Universal Robots PolyScope program: TEST_SUB_106C.urp

Program TEST_SUB_106C (installation=GD directory=/programs/GD createdIn=5.13.0 lastSavedIn=5.13.0 robotSerialNumber=20205000017)
Calibrated DH parameters: a=[-0.000157, -0.56303, -0.236706, -0.000074, -0.000109, 0]; d=[0.181705, 47.632387, 369.599619, -417.058513, 0.119878, 0.115667]; alpha=[1.570881, -0.005074, -0.001247, 1.56886, -1.570997, 0]; deltaTheta=[0, -0.405485, 5.544791, 1.143886, -0.000009, -0.000001]
InitVariablesNode
BeforeStart
  prg_no := 0
  Script file /programs/GD/CONTROL/ALIGN_AXIS.script
    | def GET_NORM_VEC(p,axis=2):
    |   rot=p[0.0, 0.0, 0.0, p[3], p[4], p[5]]
    |   vec=p[0.0, 0.0, 0.0, 0.0, 0.0, 0.0]
    |   vec[axis]=1.0
    |   norm_p=pose_trans(rot,vec)
    |   return [norm_p[0], norm_p[1], norm_p[2]]
    | end
    | 
    | def GET_INNER_PRODUCT(v1,v2):
    |   return v1[0]*v2[0]+v1[1]*v2[1]+v1[2]*v2[2]
    | end
    | def GET_OUTER_PRODUCT(v1,v2):
    |   x=v1[1]*v2[2]-v1[2]*v2[1]
    |   y=v1[2]*v2[0]-v1[0]*v2[2]
    |   z=v1[0]*v2[1]-v1[1]*v2[0]
    |   return [x,y,z]
    | end
    | def GET_THETA(v1,v2):
    | #  cos=GET_INNER_PRODUCT(v1,v2) / norm(v1) / norm(v2)
    |   cos=GET_INNER_PRODUCT(v1,v2)
    |   g_cos=cos
    |   theta=norm(acos(cos))
    |   return theta
    | end
    | 
    | def GET_ALIGNED_POSE(target,feature,axis=2):
    |   feature_from_target=pose_trans(pose_inv(target),feature)
    |   g_f_from_t=feature_from_target
    |   nz_feature_from_target=GET_NORM_VEC(feature_from_target,axis)
    |   g_nz_f_from_t=nz_feature_from_target
    |   nz_target_from_target=[0.0, 0.0, 0.0]
    |   nz_target_from_target[axis]=1.0
    |   g_nz_t_from_t=nz_target_from_target
    | 
    |   theta=GET_THETA(nz_feature_from_target,nz_target_from_target)
    |   g_theta=theta
    |   rot_vec_n=normalize(GET_OUTER_PRODUCT(nz_target_from_target,nz_feature_from_target))
    | 
    |   if theta>d2r(90.0):
    |     theta=theta-d2r(180.0)
    |   end
    |   rot_vec=rot_vec_n * (theta)
    |   rot_p=p[0.0,0.0,0.0,rot_vec[0],rot_vec[1],rot_vec[2]]
    |   return pose_trans(target,rot_p)
    | end
    | def GET_ALIGNED_TCP(feature,axis=2):
    |   tcp=get_actual_tcp_pose()
    |   return GET_ALIGNED_POSE(tcp,feature,axis)
    | end
  Script file /programs/GD/CONTROL/CYCLE_CONTROL.script
    | def GET_REG(prg_no):
    |   WorkPosNo=read_input_integer_register(4)-1                       # GPII_WorkPosNo
    |   CaptIndex[WorkPosNo]=read_input_integer_register(21)-1           # GPII_CaptColNo
    |   CaptRowNo=read_input_integer_register(20)-1        # GPII_CaptRowNo
    |   CaptStepZ=read_input_integer_register(6) / 1000.0         # GPII_CaptStepZ
    |   ReCaptNo=0
    |   if (prg_no==1203):
    |     ReCaptNo=read_input_integer_register(22)                # GPII_ReCaptNo
    |   end
    |   ReCaptZ=read_input_integer_register(7) / 1000.0         # GPII_ReCaptZ
    |   CutOffZDef=read_input_integer_register(11) / 1000.0          # GPII_CutOffZ
    |   CrankDepthFull=read_input_integer_register(10) / 1000.0   # GPII_FullDepth
    | end
    | 
    | def POSE_SUB(p, teach_frame):
    |   return pose_trans(inv(teach_frame), p)
    | end
    | 
    | def GET_BUCKET_UPPER(pos=0):
    |   if UseNewCaptPos:
    |     p=POSE_SUB(CaptPoint_C, BucketM)
    |     pX=[BKWidth/2,CaptPointL_dX,BKWidth-CaptPointR_dX]
    |     p[0]=pX[pos]
    |   else:
    |     captpos=[CaptPoint_C,CaptPoint_L,CaptPoint_R]
    |     p=captpos[pos]
    |     p=POSE_SUB(p, BucketM)
    |   end
    |   return p
    | end
    | 
    | def SET_BUCKET_DEF():
    |   BucketM=pBucketM
    |   if (WorkPosNo<0):
    |     Bucket=pBucketC
    |   else:
    |     Bucket=pBucket[WorkPosNo]
    |   end
    | end
    | 
    | def SET_BUCKET():
    |   SET_BUCKET_DEF()
    |   Bucket[2]=Bucket[2]-CaptStepZ*CaptRowNo
    | end
    | 
    | def SET_CV():
    |   CV=pCV
    | end
    | 
    | def SET_CAPT_INDEX():
    |   CaptIndexWk=CaptIndex[WorkPosNo]
    |   ReCaptZWk=0
    |   if (prg_no==1203):
    |     if   (ReCaptNo==0):
    |       if (CaptIndexWk==0):
    |         if (0<=DistPillarBak):
    |           CaptIndexWk=1
    |         else:
    |           CaptIndexWk=2
    |         end
    |         ReCaptZWk=0
    |       else:
    |         CaptIndexWk=0
    |         ReCaptZWk=0
    |       end
    |     elif (ReCaptNo==1):
    |       if (CaptIndexWk==0):
    |         CaptIndexWk=0
    |         ReCaptZWk=-ReCaptZ
    |       else:
    |         CaptIndexWk=CaptIndexWk
    |         ReCaptZWk=-ReCaptZ
    |       end
    |     else:
    |       if (CaptIndexWk==0):
    |         CaptIndexWk=0
    |         ReCaptZWk=ReCaptZ
    |       else:
    |         CaptIndexWk=CaptIndexWk
    |         ReCaptZWk=ReCaptZ
    |       end
    |     end
    |   end
    | end
    | 
    | def GET_CAPTPOS():
    |   SET_BUCKET()
    |   SET_CAPT_INDEX()
    |   if UseNewCaptPos:
    |     p=GET_BUCKET_UPPER(CaptIndexWk)
    |     p[2]=p[2]-ReCaptZWk
    |   else:
    |     captpos=[CaptPoint_C,CaptPoint_L,CaptPoint_R]
    |     p=captpos[CaptIndexWk]
    |     p[2]=p[2]-ReCaptZWk
    |     p=POSE_SUB(p, BucketM)
    |   end
    |   return p
    | end
    | 
    | def CHECK_CAPTPOS():
    |   isOK=((CaptStepZ*(read_input_integer_register(20)-1)) < (read_input_integer_register(9) / 1000.0))
    |   return isOK
    | end
    | 
    | def GET_ZSLIDE_POS(p):
    |   p[2]=p[2]-CaptStepZ*CaptRowNo
    |   return p
    | end
    | 
    | def END_CYCLE():
    |   stopl(1.2)
    |   end_force_mode()
    |   end_freedrive_mode()
    |   socket_close(socket_name)
    | end
    | 
    | def CHECK_SPEED(smax,f=[1,1,1,1,1,1]):
    |   s=TCPSpeed
    |   i=0
    |   while (i<6):
    |     if ((f[i]==1) and (smax[i]<s[i])):
    |       return False
    |     end
    |     i=i+1
    |   end
    |   return True
    | end
  Script file /programs/GD/CONTROL/ZONE_CONTROL.script
    | def GET_DIST(P1, P2):
    |   return pose_dist(P1, P2)
    | end
    | def CHECK_DIST_NEAR(P1, P2, th):
    |   return (GET_DIST(P1, P2) < th)
    | end
    | def DIST_HOME():
    |   return pose_dist(gHome_Position,CurrPos_p)
    | end
    | 
    | def CHECK_HOME():
    |   return (DIST_HOME()<ZoneDistTh)
    | end
    | 
    | def DIST_CVUpper():
    |   if (read_input_integer_register(4)==1):
    |     p=g2GD_pos1
    |   else:
    |     p=g1GD_pos1
    |   end
    |   return pose_dist(p,CurrPos_p)
    | end
    | 
    | def CHECK_CVUpper():
    |   return (DIST_CVUpper()<ZoneDistTh)
    | end
    | 
    | def CHECK_RB_POS(prg_no):
    |   ret=True
    |   if (prg_no==1001):
    |     ret=CHECK_EVAC()
    |   end
    |   if ((prg_no==1201) or (prg_no==1401) or (prg_no==1402) or (prg_no==6001) or (prg_no==6101) or (prg_no==6401) or (prg_no==6102) or (prg_no==7001)):
    |     ret=CHECK_HOME()
    |   end
    |   if ((prg_no==1002) or (prg_no==1241) or (prg_no==1261)):
    |     ret=CHECK_BKInside()
    |   end
    |   if (prg_no==1251):
    |     ret=(CHECK_HOME() or CHECK_CVUpper())
    |   end
    |   if (ret != True):
    |     SubPrgResult=801
    |     sleep(999999.0)
    |   end
    | end
    | 
    | def DIST_ORIGIN():
    |   p=CurrPos_p
    |   o=p
    |   o[0]=0.0
    |   o[1]=0.0
    |   return pose_dist(o,p)
    | end
    | 
    | def CHECK_EVAC_ORG():
    |   return (EvacRadiusTh<DIST_ORIGIN())
    | end
    | 
    | def CHECK_EVAC_X():
    |   return (EvacXTh[0]<CurrPos_p[0] and CurrPos_p[0]<EvacXTh[1])
    | end
    | 
    | def CHECK_EVAC_Y():
    |   return (EvacYTh[0]<CurrPos_p[1] and CurrPos_p[1]<EvacYTh[1])
    | end
    | 
    | def CHECK_EVAC_Z():
    |   return (EvacZTh[0]<CurrPos_p[2])
    | end
    | 
    | def CHECK_EVAC():
    |   ret=True
    |   ret=(ret and CHECK_EVAC_ORG())
    |   ret=(ret and CHECK_EVAC_X())
    |   ret=(ret and CHECK_EVAC_Y())
    |   ret=(ret and CHECK_EVAC_Z())
    |   return ret
    | end
    | 
    | def CHECK_BKInside():
    |   ret=True
    |   pos=read_input_integer_register(4)
    |   if (pos>2):
    |     ret=False
    |   else:
    |     if (not read_input_boolean_register(13+pos)):
    |       ret=False
    |       ver_3=read_input_boolean_register(13+pos)
    |     else:
    |       bk=pBucket[pos-1]
    |       if (pos==1):
    |         ret=(ret and CurrPos_p[0]>ZoneHomeX)
    |         ret=(ret and bk[1]-(BucketWidth-ZoneBucketGap)<CurrPos_p[1] and CurrPos_p[1]<bk[1]-ZoneBucketGap)
    |       elif (pos==2):
    |         ret=(ret and CurrPos_p[0]<-ZoneHomeX)
    |         ret=(ret and bk[1]+ZoneBucketGap<CurrPos_p[1] and CurrPos_p[1]<bk[1]+(BucketWidth-ZoneBucketGap))
    |       end
    |     end
    |   end
    |   return ret
    | end
    | 
    | def CHECK_CVOutside():
    |   ret=True
    |   ret=(ret and gCV_11_M[0]-Zone6ThX<CurrPos_p[0])
    |   ret=(ret and CurrPos_p[0]<gCV_11_M[0]+Zone6ThX)
    |   ret=(ret and gCV_11_M[1]-Zone6ThY<CurrPos_p[1])
    |   ret=(ret and CurrPos_p[1]<gCV_11_M[1]+Zone6ThY)
    |   return (not ret)
    | end
    | 
    | def CHECK_ZONE(no):
    |   if (no==1):
    |     return (CurrPos_p[2]>=Zone1ZTh)
    |   elif (no==2):
    |     return (CurrPos_p[0]>ZoneHomeX)
    |   elif (no==3):
    |     return (CurrPos_p[0]<-ZoneHomeX)
    |   elif (no==4):
    |     return CHECK_CVUpper()
    |   elif (no==5):
    |     return CHECK_BKInside()
    |   elif (no==6):
    |     return CHECK_CVOutside()
    |   end
    | end
  Script file /programs/GD/CONTROL/ROTATE_CONTROL.script
    | def GET_TCP_FORCE_TOOL():
    |   force_torque=get_tcp_force()
    |   force_B=p[force_torque[0], force_torque[1], force_torque[2], 0, 0, 0]
    |   torque_B=p[force_torque[3], force_torque[4], force_torque[5], 0, 0, 0]
    |   tcp=get_actual_tcp_pose()
    |   rotation_BT=p[0, 0, 0, tcp[3], tcp[4], tcp[5]]
    |   force_T=pose_trans(pose_inv(rotation_BT), force_B)
    |   torque_T=pose_trans(pose_inv(rotation_BT), torque_B)
    |   force_torque_T=p[force_T[0], force_T[1], force_T[2], torque_T[0], torque_T[1], torque_T[2]]
    |   return force_torque_T
    | end
    | 
    | def CHECK_VALUE_RZ():
    |   return True
    | end
    | 
    | def GET_FORCE_VALUE_RZ(target):
    |   PoseSub= pose_sub (CurrPos_p,target)
    |   RYSub=r2d(PoseSub[4])
    |   RZSub=r2d(PoseSub[5])
    | #  if (RYSub<RZSupRYRange[0] or RZSupRYRange[1]<RYSub):
    | #    RZSupForceVal=0.0
    | #    return RZSupForceVal
    | #  end
    |   if (RZSub<0):
    |     RZMin=RZSupDegMin[0]
    |     RZRatio=RZSupRatio[0]
    |     RZOffset=RZSupOffset[0]
    |   else:
    |     RZMin=RZSupDegMin[1]
    |     RZRatio=RZSupRatio[1]
    |     RZOffset=-RZSupOffset[1]
    |   end
    |   if (norm(RZSub) >= norm(RZMin)):
    |     RZSupForceVal=(RZMin-RZSub)*RZRatio+RZOffset
    |   else:
    |     RZSupForceVal=0
    |   end
    |   if (RZSupForceVal<RZSupForceRange[0]):
    |     RZSupForceVal=RZSupForceRange[0]
    |   elif (RZSupForceRange[1]<RZSupForceVal):
    |     RZSupForceVal=RZSupForceRange[1]
    |   end
    |   if (RYSub<RZSupRYRange[0] or RZSupRYRange[1]<RYSub):
    |     RZSupForceVal=0
    |   end
    |   if ((not UseRZSupStep1) and (ForceStep==1)):
    |     RZSupForceVal=0
    |   end
    |   return RZSupForceVal
    | end
    | 
    | def GET_CVCORR_VALUE(target):
    |   PoseSub=pose_sub(CurrPos_p,target)
    |   RYSub=r2d(PoseSub[4])
    |   CVCorrRYSub=RYSub
    |   if (RYSub<0):
    |     RYMin=-CVCorrDegMin[0]
    |     RZRatio=CVCorrRatio[0]
    |     RZOffset=-CVCorrOffset[0]
    |   else:
    |     RYMin=-CVCorrDegMin[1]
    |     RZRatio=CVCorrRatio[1]
    |     RZOffset=CVCorrOffset[1]
    |   end
    |   if (norm(RYSub) >= norm(RYMin)):
    |     t=get_tcp_offset()
    |     CVCorrYVal=-t[2]*sin(d2r(RYSub))
    |     CVCorrRZVal=RYSub*RZRatio+RZOffset
    |   else:
    |     CVCorrYVal=0
    |     CVCorrRZVal=0
    |   end
    | end
    | 
    | def GET_CVCORR_POS(target):
    |   pos= pose_add (p[0,0,0,0,0,d2r(-CVCorrRZVal)],p[0,0,0,target[3],target[4],target[5]])
    |   pos=p[target[0],target[1],target[2],pos[3],pos[4],pos[5]]
    |   return pos
    | end
Robot Program (runOnlyOnce=true)
  SuppressedNode
    Wait Sleep waitTime=20
  If UseCutOffTCP
    Set NoAction tcp=TCP_1
    CutOffPos := p[0.,0.,0.,0.,0.,0.]
    CutOffPos := GET_ALIGNED_TCP(CutOffPos)
    Script: CurrPos=get_actual_tool_flange_pose()
    CutOffTCP := pose_trans(pose_inv(CurrPos),CutOffPos)
    SuppressedNode
      MoveJ speed 60 deg/s, acceleration 80 deg/s^2 (useActiveTCP=true) feature=Base
        Waypoint Variable (Variable): variable=CutOffPos
    Set NoAction tcp=ZERO
    CutOffTCP := pose_trans(get_tcp_offset(),CutOffTCP)
    Set NoAction tcp=TCP_1
  Else 
    Set NoAction tcp=TCP_1
    CutOffTCP := get_tcp_offset()
  Script: set_tcp(CutOffTCP)
  MoveL speed 250 mm/s, acceleration 50 mm/s^2 (useActiveTCP=true) feature=Base
    If UseZSlide
      gGD_pos5 := GET_ZSLIDE_POS(g1GD_pos5_NEAR)
    Else 
      gGD_pos5 := g1GD_pos5
    SuppressedNode
      Folder CV_CORR_RZ
        If UseCVCorr
          RZSub := CVCorrRZVal
          Set NoAction tcp=TCP_1
          Wait Sleep waitTime=0.02
          SuppressedNode
            Script: CurrPos_p=get_actual_tcp_pose()
          Script: CurrPos_p=gGD_pos5
          SuppressedNode
            Script: CurrPos_p[2]=CurrPos_p[2]-0.45
          MoveL speed 60 mm/s, acceleration 10 mm/s^2 (useActiveTCP=false) tcp=TCP_1; feature=Base
            PoseAdd := pose_add(p[0,0,0,0,0,d2r(-RZSub)],p[0,0,0,CurrPos_p[3],CurrPos_p[4],CurrPos_p[5]])
            PoseAdd := p[CurrPos_p[0],CurrPos_p[1],CurrPos_p[2],PoseAdd[3],PoseAdd[4],PoseAdd[5]]
            Waypoint Variable (Variable): variable=PoseAdd
    Script: DistBKUpper=GET_DIST(CurrPos_p,gGD_pos5)
    If ( not CHECK_DIST_NEAR(CurrPos_p, gGD_pos5, DistBKUpperTh))
      Waypoint Variable (Variable): variable=gGD_pos5
  MoveL speed 400 mm/s, acceleration 140 mm/s^2 (useActiveTCP=true) feature=Base
    SetPayload (workpieceName=k10)
    Waypoint Variable (Variable): variable(featureName=g1GD_pos3)
    Waypoint Variable (Variable): variable(featureName=g1GD_pos2)
  MoveL speed 400 mm/s, acceleration 140 mm/s^2 (useActiveTCP=true) feature=Base
    SetPayload (workpieceName=k120)
    Waypoint Variable (Variable): motionParameters(blendRadius=0.1); variable(featureName=g1GD_pos1)
    If UseCVCorr
      PoseAdd := GET_CVCORR_POS(g1GD_pos1)
      Waypoint Variable (Variable): variable=PoseAdd
  MoveJ speed 20 deg/s, acceleration 40 deg/s^2 (useActiveTCP=false) tcp=TCP_1; feature=Base
    Waypoint Variable (Variable): variable(featureName=gHome_Position)
Thread スレッド_2 (runOnlyOnce=false)
  Script: CurrPos=get_actual_tool_flange_pose()
  Script: CurrPos_p=get_actual_tcp_pose()
  Script: Currpos_p_UF0=pose_trans(pose_inv(UF), CurrPos_p)
  TCPSpeed := get_actual_tcp_speed()
  TCPForce := get_tcp_force()
  Script: sync()
